Staubli VAL3: constantes.pjx

--- constantes.pjx ---
Parameters version=s7.6.3 stackSize=5000 millimeterUnit=true
Program file=init.pgx
Program file=start.pgx
Program file=stop.pgx
Data file=constantes.dtx

--- constantes.dtx ---
mdesc mNomSpeed
public num nDRV_ACTIV
public num nRdy2SwitchON
public num nSwitchONDis
public num nNotRdySwiON
public num nSwitchedON
public num nOperatEnabled
public num nQuickStopActiv
public num nFaultReacActiv
public num nFaultState
public num nDRV_FAULT
num nEtapeInit
public num nNOTEXIST
public num nAXIS7
public num nAXIS8 = 1
public num nDEBUGDRIVE = 1
public num nHWALM_TESTHW
public num nHWALM_FEEDPW
public num nHWALM_UDRVOLT
public num nHWALM_OVRVOLT
public num nHWALM_OVRCUR
public num nHWALM_TEMPDIS
public num nHWALM_FRENO
public num nHWALM_EEPROM
public num nHWALM_FUSE5VLT
public num nHWALM_THERMMOT
public num nHWALM_HALL
public num nHWALM_TRANSDUC
public num nHWALM_CONNMOT
public num nSWALM_FUNGO
public num nSWALM_TAGLIA
public num nSWALM_CSDATI
public num nSWALM_I2T
public num nSWALM_POSITION
public num nSWALM_ENCODER
public num nSWALM_HALLENC
public num nSWALM_OVRSPEED
public num nSWALM_TRANSDUC
public num nSWALM_ENCMASTR
public num nSWALM_UDRVOLT
public num nSWALM_POSROTOR
public num nSWALM_OFFSREF
public num nSWALM_I2TREGEN
public num nSWALM_CANBUS
public num nSTATUS_REMOTE
public num nHOMINGMODE = 6
public num nINTERPMODE = 7
public num nTO_DRVENABLE
public num nTO_DRVDISABLE
public num nPPMODE

--- START.PGX ---
program start()
begin


end

--- INIT.PGX ---
public program init()
begin
  //该库相当于一纯数据变量库,用于Sample,extAxisCan数据交换
  // **************************************
  // *****        DRIVE STATES        *****
  // **************************************
  // refer to CiA draft proposal 402 page 51 (协议402,51页)
  //根6041，驱动器正常激活时，0-3, 5 and 6 位1，换成十进制为111dec=1101111bin
  // -- Value for binary masking bits 0-3, 5 and 6

  nDRV_ACTIV=111
  //
  // -- Value for binary masking bits 0-3 and 6
  //100 1111
  nDRV_FAULT=79

  //以下位外部驱动器状态（6041）
  // --not Ready to switch on
  nNotRdySwiON=0

  // -- Switch on disabled 100 0000
  nSwitchONDis=64

  // -- ready to switch ON
  //10 0001
  nRdy2SwitchON=33

  // -- Switched ON 10 0011

  nSwitchedON=35

  //-- Operation enabled 10 0111
  nOperatEnabled=39
  // -- Quick stop active  0111
  nQuickStopActiv=7

  // Fault reaction active 1111
  nFaultReacActiv=15

  // -- Fault state 1000
  nFaultState=8

  // *******************************************
  // *****    HARDWARE DRIVE ALARMS        *****
  // *******************************************
  // -- System test failed (RAM or ADC or internal device malfunction
  nHWALM_TESTHW= 1
  // -- Power failure
  nHWALM_FEEDPW= 2
  // -- Bus under-voltage. The lower threshold (80VDC) has been underpassed
  nHWALM_UDRVOLT=4
  // -- Bus over-voltage. The highest Treshold (630VDC) has been overpassed
  nHWALM_OVRVOLT=8
  // -- Over current
  nHWALM_OVRCUR=16
  // -- Heat sink temperature failed (Tc>80°C)
  nHWALM_TEMPDIS=32
  // -- Clamp circuit failure.
  nHWALM_FRENO=64
  // -- EEPROM checksulm failure
  nHWALM_EEPROM=128
  // -- FUSE 5 VOLT failure on transducer line
  nHWALM_FUSE5VLT=256
  // -- Motor thermal protection failure
  nHWALM_THERMMOT=512
  // -- Hall effects wrong configuration detected
  nHWALM_HALL=1024
  // -- Transducer hardware failure
  nHWALM_TRANSDUC=2048
  // -- Phase motor current unbalanced
  nHWALM_CONNMOT=4096

  // *******************************************
  // *****    SOFTWARE DRIVE ALARMS        *****
  // *******************************************
  // -- customized FAIL (not used)
  nSWALM_FUNGO = 1
  // -- drive size is not coherent
  nSWALM_TAGLIA=2
  // -- EEPROM checksum failure
  nSWALM_CSDATI=4
  // -- Canbus communication failure
  nSWALM_CANBUS=8
  // -- Position loop failure (following error,overtravel....)
  nSWALM_POSITION=16
  // -- I2T protection
  nSWALM_I2T=32
  // -- Maximum speed exceeded (parameter velMax)
  nSWALM_OVRSPEED=64
  // -- Hall efect and encoder checksum failure
  nSWALM_HALLENC=128
  // -- encoder zero tag out of position or missing.
  nSWALM_ENCODER=256
  // -- Transducer failure (resolver oder enDat)
  nSWALM_TRANSDUC=512
  // -- Master encoder zero tag out
  nSWALM_ENCMASTR=1024
  // -- Bus under-voltage
   nSWALM_UDRVOLT=2048
  // -- Sensorless rotor phasing procedure failure
  nSWALM_POSROTOR=4096
  // -- Speed reference automatic offset compensation failure
  nSWALM_OFFSREF=8192
  // -- I2T protection for clamp resistor failure
  nSWALM_I2TREGEN=16384

  //
  // value for not existing val3 task
  nNOTEXIST=-1
  nDEBUGDRIVE=1
  // 电机remote状态位
  nSTATUS_REMOTE=0

  // 使电机使能的时间
  nTO_DRVENABLE=2
  // 电机去使能的时间
  nTO_DRVDISABLE=2

  //驱动器模式
  nHOMINGMODE = 6
  nINTERPMODE=7
  nPPMODE=1
end
